(*
SPDX-FileCopyrightText: © 2026 Oleksandr Tiutyk <trofimich@gmail.com>
SPDX-License-Identifier: MIT
License: https://opensource.org/license/mit
*)

(*!
<summary>Base class for composite activities that execute at most one child activity at a time.</summary>
<description>
Provides state translation helpers for mapping a child activity's state into the parent composite's running,
stopping or resetting result, as well as single-parent attachment validation and child resetting.
</description>
*)

{attribute 'no_explicit_call' := 'do not call this function block directly'}
FUNCTION_BLOCK ABSTRACT ExclusiveCompositeActivity EXTENDS Activity
	IMPLEMENTS IExclusiveCompositeActivity

(*!
<summary>Returns the currently selected child activity, or 0 when no child is selected.</summary>
*)
{attribute 'monitoring' := 'call'}
PROPERTY ABSTRACT CurrentActivity : IActivity
GET
END_GET
END_PROPERTY

(*!
<summary>Translates a child activity state after a reset step into the parent composite's resetting result.</summary>
<description>
ACTIVE_RESETTING and ACTIVE_CANCELLING map to WORK_IN_PROGRESS. PASSIVE_READY maps to WORK_RESET. Any other
state raises InvalidNestedWorkflowStateException.
</description>
<param name="childState">Observed state of the child activity being reset.</param>
*)
METHOD PROTECTED MapChildResettingState : ACTIVITY_RESETTING_STATE
VAR_INPUT
	childState : WORKFLOW_ELEMENT_STATE;
END_VAR
VAR
END_VAR
CASE childState OF
	WORKFLOW_ELEMENT_STATE.ACTIVE_RESETTING,
	WORKFLOW_ELEMENT_STATE.ACTIVE_CANCELLING:
		MapChildResettingState := ACTIVITY_RESETTING_STATE.WORK_IN_PROGRESS;

	WORKFLOW_ELEMENT_STATE.PASSIVE_READY:
		MapChildResettingState := ACTIVITY_RESETTING_STATE.WORK_RESET;

	ELSE
		WorkflowExceptions.ThrowInvalidNestedWorkflowState(
			sourceNamespaceName := NamespaceName,
			sourceClassName := ClassName,
			sourcePOUName := __POUNAME(),
			sourcePosition := __POSITION(),
			nestedActivityState := childState
		);
END_CASE
END_METHOD

(*!
<summary>Translates a child activity state after a running step into the parent composite's running result.</summary>
<description>
ACTIVE_RUNNING maps to WORK_IN_PROGRESS, PASSIVE_COMPLETED to WORK_COMPLETED, and PASSIVE_HALTED to
WORK_HALTED. Any other state raises InvalidNestedWorkflowStateException.
</description>
<param name="childState">Observed state of the active child activity.</param>
*)
METHOD PROTECTED MapChildRunningState : ACTIVITY_RUNNING_STATE
VAR_INPUT
	childState : WORKFLOW_ELEMENT_STATE;
END_VAR
VAR
END_VAR
CASE childState OF
	WORKFLOW_ELEMENT_STATE.ACTIVE_RUNNING:
		MapChildRunningState := ACTIVITY_RUNNING_STATE.WORK_IN_PROGRESS;

	WORKFLOW_ELEMENT_STATE.PASSIVE_COMPLETED:
		MapChildRunningState := ACTIVITY_RUNNING_STATE.WORK_COMPLETED;

	WORKFLOW_ELEMENT_STATE.PASSIVE_HALTED:
		MapChildRunningState := ACTIVITY_RUNNING_STATE.WORK_HALTED;

	ELSE
		WorkflowExceptions.ThrowInvalidNestedWorkflowState(
			sourceNamespaceName := NamespaceName,
			sourceClassName := ClassName,
			sourcePOUName := __POUNAME(),
			sourcePosition := __POSITION(),
			nestedActivityState := childState
		);
END_CASE
END_METHOD

(*!
<summary>Translates a child activity state after a stopping step into the parent composite's stopping result.</summary>
<description>
ACTIVE_CANCELLING and ACTIVE_SUSPENDING map to WORK_IN_PROGRESS; PASSIVE_CANCELLED and PASSIVE_SUSPENDED map
to WORK_STOPPED; PASSIVE_COMPLETED maps to WORK_COMPLETED; PASSIVE_HALTED maps to WORK_HALTED. Any other state
raises InvalidNestedWorkflowStateException.
</description>
<param name="childState">Observed state of the stopping child activity.</param>
*)
METHOD PROTECTED MapChildStoppingState : ACTIVITY_STOPPING_STATE
VAR_INPUT
	childState : WORKFLOW_ELEMENT_STATE;
END_VAR
VAR
END_VAR
CASE childState OF
	WORKFLOW_ELEMENT_STATE.ACTIVE_CANCELLING, WORKFLOW_ELEMENT_STATE.ACTIVE_SUSPENDING:
		MapChildStoppingState := ACTIVITY_STOPPING_STATE.WORK_IN_PROGRESS;

	WORKFLOW_ELEMENT_STATE.PASSIVE_CANCELLED, WORKFLOW_ELEMENT_STATE.PASSIVE_SUSPENDED:
		MapChildStoppingState := ACTIVITY_STOPPING_STATE.WORK_STOPPED;

	WORKFLOW_ELEMENT_STATE.PASSIVE_COMPLETED:
		MapChildStoppingState := ACTIVITY_STOPPING_STATE.WORK_COMPLETED;

	WORKFLOW_ELEMENT_STATE.PASSIVE_HALTED:
		MapChildStoppingState := ACTIVITY_STOPPING_STATE.WORK_HALTED;

	ELSE
		WorkflowExceptions.ThrowInvalidNestedWorkflowState(
			sourceNamespaceName := NamespaceName,
			sourceClassName := ClassName,
			sourcePOUName := __POUNAME(),
			sourcePosition := __POSITION(),
			nestedActivityState := childState
		);
END_CASE
END_METHOD

(*!
<summary>Advances resetting of a child activity toward PASSIVE_READY by one step.</summary>
<description>
Returns WORK_RESET immediately when childActivity is 0 or already in PASSIVE_READY. If the child was left in
PASSIVE_SUSPENDED or ACTIVE_CANCELLING, drives cancellation to PASSIVE_CANCELLED before invoking RequestReset.
In ACTIVE_RESETTING, advances the child via Execute; in finished passive states, invokes RequestReset.
</description>
<param name="childActivity">Child activity to reset, or 0.</param>
*)
METHOD PROTECTED ResetChildActivity : ACTIVITY_RESETTING_STATE
VAR_INPUT
	childActivity : IActivity;
END_VAR
ResetChildActivity := WorkflowElementHelper.ResetChildActivity(
	childActivity := childActivity,
	cancelReason := "Parent composite activity resetting",
	sourceClassName := ClassName,
	sourcePOUName := __POUNAME()
);
END_METHOD

(*!
<summary>
Verifies that a candidate child activity can be attached to this composite without cycles or shared parents.
</summary>
<description>
Delegates to Workflows.ValidateElementAttachment for readiness, cycles, existing parent, root exclusion and
fixed workflow association. Reusing the same link during Configure is allowed; append methods must reject
occupied slots separately. No topology or ownership mutation is performed.
</description>
<param name="childActivity">Candidate child activity to validate.</param>
<param name="argumentName">Parameter name for diagnostic reporting.</param>
*)
METHOD PROTECTED ValidateChildActivityAttachment
VAR_INPUT
	childActivity : IActivity;
	argumentName : STRING(255);
END_VAR
WorkflowElementHelper.ValidateChildActivityAttachment(
	parent := THIS^,
	childActivity := childActivity,
	argumentName := argumentName,
	sourceClassName := ClassName,
	sourcePOUName := __POUNAME()
);
END_METHOD

END_FUNCTION_BLOCK

(* stored: Version 1.1.0.1
   POU ExclusiveCompositeActivity: Id {13ce720f-cc4b-4c1a-8e26-2a31330dfb74}, SpecialFunc None
   Folder Service methods: Id {760a10bf-9189-41b6-af5c-f9a53d374520}
   Property CurrentActivity: Id {f87026db-b40e-41a2-b4b1-af04873341d9}
   Get Get: Id {16b243ca-e41f-4cab-b539-f522d3ba872b}
   Method MapChildResettingState: Id {3c7f81d1-2b46-4c60-9d21-4e7782e66b10}
   Method MapChildRunningState: Id {c15358dd-5baf-4122-b6b7-ff0ce4db1cb4}
   Method MapChildStoppingState: Id {1b24d1c5-0190-4a91-b76b-ad26fb99c654}
   Method ResetChildActivity: Id {5b6c11e9-473a-41b3-9f90-2e5779ca1841}
   Method ValidateChildActivityAttachment: Id {8a41e822-91f2-4b4e-83f4-650830f291c3} *)
